FUNCTION_BLOCK DATA_AGGREGATOR
  {SET_ATTRIBUTE(OpcUa, SERVICE)}
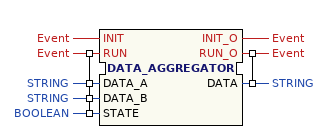
  EVENT_INPUT
    INIT;
    RUN WITH DATA_A, DATA_B, STATE;
  END_EVENT
  EVENT_OUTPUT
    INIT_O;
    RUN_O WITH DATA;
  END_EVENT
  VAR_INPUT
    DATA_A : STRING;
    DATA_B : STRING;
    STATE : BOOLEAN;
  END_VAR
  VAR_OUTPUT
    DATA : STRING;
  END_VAR
END_FUNCTION_BLOCK
